(* PLC project Infinite State Machine Library, CODESYS CODESYS V3.5 SP21 Patch 2, author Roy Ratcliffe *)
(* stored: creationDateTime 2025-10-15T13:16:43.0309977, version 0.1.1.1, modificationDateTime 2025-09-09T17:58:13.641387, organization Roy Ratcliffe *)

TYPE IStateArray : ARRAY[0..ISM.gc_iMaxDepth] OF IState;
END_TYPE

{attribute 'qualified_only'}
VAR_GLOBAL CONSTANT  (* ISM *)
  gc_iMaxDepth : INT := 7;
END_VAR

INTERFACE IState
METHOD Enter
  VAR_INPUT
    fbStateMachine : StateMachine;
  END_VAR
END_METHOD
METHOD Leave
  VAR_INPUT
    fbStateMachine : StateMachine;
  END_VAR
END_METHOD
PROPERTY SuperState : IState
END_PROPERTY
END_INTERFACE

FUNCTION_BLOCK StateMachine
  VAR
    itfStates : IStateArray;
    iDepth : INT := 0;
  END_VAR

            
          

METHOD Jump
  VAR_INPUT
    itfState : IState;
  END_VAR
                  iDepth := DepthOfState(itfState, ISM.gc_iMaxDepth, itfStates);

                
END_METHOD

METHOD Top : IState
                  IF iDepth > 0 THEN
	Top := itfStates[iDepth - 1];
END_IF

                
END_METHOD

METHOD Push : BOOL
  VAR_INPUT
    itfState : IState;
  END_VAR
                  Push := iDepth < ISM.gc_iMaxDepth;
IF Push THEN
	itfStates[iDepth] := itfState;
	iDepth := iDepth + 1;
END_IF

                
END_METHOD

METHOD Pop : IState
                  IF iDepth > 0 THEN
	iDepth := iDepth - 1;
	Pop := itfStates[iDepth];
    (*
     * Clear the popped state from the stack. This is not strictly necessary,
     * but it can help catch use-after-free bugs.
     *)
	itfStates[iDepth] := 0;
ELSE
	Pop := 0;
END_IF

                
END_METHOD

METHOD GoTo
  VAR_INPUT
    itfState : IState;
  END_VAR
  VAR
    fbStateMachine : StateMachine;
    iDepth : INT := 0;
  END_VAR
                  fbStateMachine.Jump(itfState);
WHILE iDepth < Depth() AND iDepth < fbStateMachine.Depth() AND IsSameState(AtLevel(iDepth), fbStateMachine.AtLevel(iDepth)) DO
	iDepth := iDepth + 1;
END_WHILE
WHILE Depth() > iDepth DO
	Leave();
END_WHILE
WHILE fbStateMachine.Depth() > iDepth DO
	Enter(fbStateMachine.AtLevel(iDepth));
	iDepth := iDepth + 1;
END_WHILE

                
END_METHOD

METHOD Depth : INT
                  Depth := iDepth;

                
END_METHOD

METHOD AtLevel : IState
  VAR_INPUT
    iLevel : INT;
  END_VAR
                  IF 0 <= iLevel AND iLevel < iDepth THEN
	AtLevel := itfStates[iLevel];
END_IF

                
END_METHOD

METHOD Enter
  VAR_INPUT
    itfState : IState;
  END_VAR
                  IF Push(itfState) THEN
	itfState.Enter(THIS^);
END_IF

                
END_METHOD

METHOD Leave
  VAR
    itfState : IState;
  END_VAR
                  itfState := Pop();
IF itfState <> 0 THEN
	itfState.Leave(THIS^);
END_IF

                
END_METHOD

METHOD In : BOOL
  VAR_INPUT
    itfState : IState;
  END_VAR
  VAR
    iLevel : INT := 0;
  END_VAR
                  (*
 * The following do-while loop's condition assumes early-out semantics.
 * It assumes that the second sub-condition does *not* evaluate unless the first sub-condition is true.
 *)
WHILE iLevel < iDepth AND itfStates[iLevel] <> itfState DO
	iLevel := iLevel + 1;
END_WHILE
In := iLevel < iDepth;

                
END_METHOD
END_FUNCTION_BLOCK

{attribute 'suppress_warning' := '0561'}
FUNCTION DepthOfState : INT
  VAR_INPUT
    itfState : IState;
    iDepth : INT;
    itfStates : REFERENCE TO IStateArray;
  END_VAR

            IF itfState = 0 THEN
	DepthOfState := 0;
ELSE
	DepthOfState := Topology(itfState, iDepth, itfStates);
END_IF

          
END_FUNCTION

FUNCTION IsSameState : BOOL
  VAR_INPUT
    itfStateLHS : IState;
    itfStateRHS : IState;
  END_VAR

            IsSameState := itfStateLHS = itfStateRHS;

          
END_FUNCTION

{attribute 'suppress_warning' := '0561'}
FUNCTION Topology : INT
  VAR_INPUT
    itfState : IState;
    iDepth : INT;
    itfStates : REFERENCE TO IStateArray;
  END_VAR

            IF iDepth = 0 THEN
	Topology := 0;
ELSE
	Topology := DepthOfState(itfState.SuperState, iDepth - 1, itfStates);
	itfStates[Topology] := itfState;
	Topology := Topology + 1;
END_IF

          
END_FUNCTION
